(* CODESYS project Motion.xml

Project tree, tasks and I/O mapping:
  program Motion [CFC]
*)

// Motion
PROGRAM Motion
VAR
END_VAR

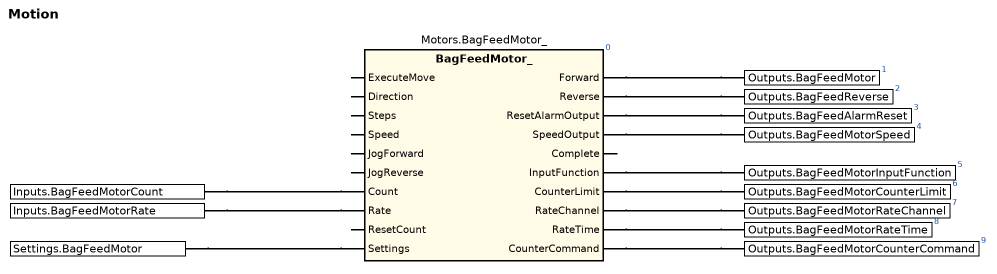
Motors.BagFeedMotor_(
    Count := Inputs.BagFeedMotorCount,
    Rate := Inputs.BagFeedMotorRate,
    Settings := Settings.BagFeedMotor); // BagFeedMotor_
Outputs.BagFeedMotor := Motors.BagFeedMotor_.Forward;
Outputs.BagFeedReverse := Motors.BagFeedMotor_.Reverse;
Outputs.BagFeedAlarmReset := Motors.BagFeedMotor_.ResetAlarmOutput;
Outputs.BagFeedMotorSpeed := Motors.BagFeedMotor_.SpeedOutput;
Outputs.BagFeedMotorInputFunction := Motors.BagFeedMotor_.InputFunction;
Outputs.BagFeedMotorCounterLimit := Motors.BagFeedMotor_.CounterLimit;
Outputs.BagFeedMotorRateChannel := Motors.BagFeedMotor_.RateChannel;
Outputs.BagFeedMotorRateTime := Motors.BagFeedMotor_.RateTime;
Outputs.BagFeedMotorCounterCommand := Motors.BagFeedMotor_.CounterCommand;

END_PROGRAM
